// TIA Portal V17 export
// export: Created 2025-06-26T07:49:49.5102857Z, ExportSetting WithDefaults, DisplayName Totally Integrated Automation Portal, DisplayVersion V17 Update 8, DisplayName TIA Portal Openness, DisplayVersion V17 Update 8, DisplayName TIA Portal Version Control Interface, DisplayVersion V17, DisplayName STEP 7 Professional, DisplayVersion V17 Update 8, DisplayName STEP 7 Safety, DisplayVersion V17 Update 6, DisplayName WinCC Advanced, DisplayVersion V17 Update 8
FUNCTION_BLOCK "fbLimitAlarm"   // FB46, FBD
{ S7_Optimized_Access := 'TRUE' }
VERSION : 0.1
// stored: AutoNumber true, IsIECCheckEnabled false, IsRetainMemResEnabled false, MemoryReserve 0, SetENOAutomatically false, UDAEnableTagReadback false
   VAR_INPUT
      fValue : Real;
      fLimit : Real;
      fHysteresis : Real;
      bType : Bool;
      tAlarmDelay : Time;
      bAck : Bool;
      bEnable : Bool;
   END_VAR
   VAR_OUTPUT
      bActive : Bool;
      bActiveUnack : Bool;
   END_VAR
   VAR
      Limit : "fbHysteresis";
      Alarm { S7_SetPoint := 'True'} : "fbAlarm";
   END_VAR
   VAR_TEMP
      AlarmCondition : Bool;
   END_VAR
BEGIN

REGION Network 1: Check for alarm condition
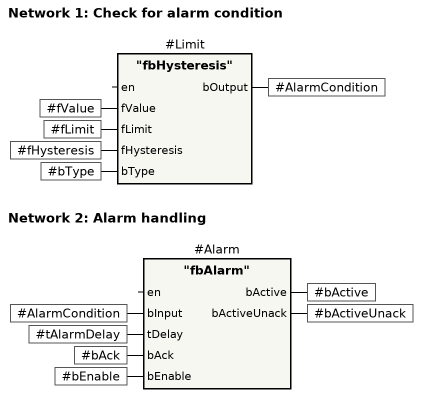
   #Limit(fValue := #fValue,   // "fbHysteresis"
          fLimit := #fLimit,
          fHysteresis := #fHysteresis,
          bType := #bType,
          bOutput => #AlarmCondition);
END_REGION

REGION Network 2: Alarm handling
   #Alarm(bInput := #AlarmCondition,   // "fbAlarm"
          tDelay := #tAlarmDelay,
          bAck := #bAck,
          bEnable := #bEnable,
          bActive => #bActive,
          bActiveUnack => #bActiveUnack);
END_REGION
END_FUNCTION_BLOCK
